TYPE "typePropOutputParam"
VERSION : 0.1
   STRUCT
      filterTimeConsts : Array[1.."AXIS_NUM"] of Real;
   END_STRUCT;

END_TYPE

